TYPE AxesIOStatuses :
STRUCT
	///Is the I/O in a healthy state?
	healthStatus: HealthStatus;
END_STRUCT
END_TYPE

(* stored: Version 1.1.0.1, ProductVersion 3.1.4019.2
   DUT AxesIOStatuses: Id {3dc038d5-cec3-45f3-b34e-0937ee33dbb2} *)
